(* IEC 61131-3 sources: RL_MAR/experiments/comparison/autoplc/results/gpt-4o_20260511_211137/med_43, 1 file *)

(* ---- med_43_1.st ---- *)
FUNCTION_BLOCK SandwichMaker
VAR_INPUT
    BreadFeeder : BOOL; (* Input: Detects the presence of bread slices *)
    Ingredient1 : BOOL; (* Input: Detects the presence of Ingredient 1 (e.g., cheese) *)
    Ingredient2 : BOOL; (* Input: Detects the presence of Ingredient 2 (e.g., lettuce) *)
    Ingredient3 : BOOL; (* Input: Detects the presence of Ingredient 3 (e.g., tomatoes) *)
    Condiment1 : BOOL; (* Input: Detects the presence of Condiment 1 (e.g., mayo) *)
    Condiment2 : BOOL; (* Input: Detects the presence of Condiment 2 (e.g., mustard) *)
END_VAR
VAR_OUTPUT
    ConveyorMotor : BOOL; (* Output: Controls the conveyor belt motor *)
    AssembleMotor : BOOL; (* Output: Controls the sandwich assembly motor *)
END_VAR
VAR
    SliceCount : INT := 0; (* Counter for bread slices *)
END_VAR

(* Initialization *)
ConveyorMotor := FALSE;
AssembleMotor := FALSE;

(* Bread Detection and Conveyor Control *)
IF BreadFeeder THEN
    ConveyorMotor := TRUE;
    SliceCount := SliceCount + 1;
ELSE
    ConveyorMotor := FALSE;
END_IF

(* Assembly Readiness Check *)
IF SliceCount >= 2 THEN
    IF Ingredient1 AND Ingredient2 AND Ingredient3 AND Condiment1 AND Condiment2 THEN
        AssembleMotor := TRUE;
    ELSE
        AssembleMotor := FALSE;
    END_IF
ELSE
    AssembleMotor := FALSE;
END_IF

END_FUNCTION_BLOCK
